{attribute 'GeneratedUsingTerminal: EJ6002-0000-0016'}
{attribute addProperty BoxType "EJ6002-0000-0016"}
{attribute addProperty Id "COM_Inputs_Channel_1AT %I*COM_Inputs_Channel_3801C95E30COM_Inputs_Channel_2AT %I*COM_Inputs_Channel_3801C95E30COM_Outputs_Channel_1AT %Q*COM_Outputs_Channel_EADA2E0D27COM_Outputs_Channel_2AT %Q*COM_Outputs_Channel_EADA2E0D27WcStateAT %I*WcState_9091E0EB2InfoDataAT %I*InfoData_94A18F5E2"}
{attribute addProperty CRC "1143283035"}
{attribute addProperty Size "118"}
TYPE EJ6002_44251D5B EXTENDS EtcSlaveTerminalBase_947E5A46 :
STRUCT
	{attribute addProperty Name "COM_Inputs_Channel_1"}
	COM_Inputs_Channel_1 : COM_Inputs_Channel_3801C95E;
	{attribute addProperty Name "COM_Inputs_Channel_2"}
	COM_Inputs_Channel_2 : COM_Inputs_Channel_3801C95E;
	{attribute addProperty Name "COM_Outputs_Channel_1"}
	COM_Outputs_Channel_1 : COM_Outputs_Channel_EADA2E0D;
	{attribute addProperty Name "COM_Outputs_Channel_2"}
	COM_Outputs_Channel_2 : COM_Outputs_Channel_EADA2E0D;
	{attribute addProperty Name "WcState"}
	WcState : WcState_9091E0EB;
	{attribute addProperty Name "InfoData"}
	InfoData : InfoData_94A18F5E;
END_STRUCT
END_TYPE

(* stored: Version 1.2.0.0, ProductVersion 3.1.4024.9
   DUT EJ6002_44251D5B: Id {e8544952-99e5-4f5c-b14c-44c7306815fb} *)
